// :Description: Example function block for TcKit parser validation.
// :param bEnable: Rising edge starts the operation
// :param nSetpoint: Target value in engineering units
FUNCTION_BLOCK FB_Example
VAR_INPUT
    bEnable    : BOOL;
    nSetpoint  : INT;
END_VAR
VAR_OUTPUT
    bDone      : BOOL;
    bError     : BOOL;
    nErrorId   : UDINT;
END_VAR
VAR
    eState     : E_ExampleState := E_ExampleState.Idle;
    nInternal  : INT;
END_VAR


CASE eState OF
    E_ExampleState.Idle:
        IF bEnable THEN
            eState := E_ExampleState.Running;
        END_IF

    E_ExampleState.Running:
        nInternal := nSetpoint;
        bDone := TRUE;
        eState := E_ExampleState.Idle;

    E_ExampleState.Error:
        bError := TRUE;
END_CASE


// :Description: Execute one cycle of the operation.
// :returns: TRUE when the operation completes successfully
METHOD Execute : BOOL
VAR_INPUT
    bTrigger : BOOL;
END_VAR

IF bTrigger THEN
    bDone := FALSE;
    bError := FALSE;
    nErrorId := 0;
    eState := E_ExampleState.Running;
END_IF

Execute := bDone;
END_METHOD


// :Description: Reset error state and outputs.
METHOD Reset : BOOL

bDone := FALSE;
bError := FALSE;
nErrorId := 0;
eState := E_ExampleState.Idle;
Reset := TRUE;
END_METHOD

END_FUNCTION_BLOCK

(* stored: Version 1.1.0.1, ProductVersion 3.1.4026.0
   POU FB_Example: Id {12345678-0000-0000-0000-000000000001}, SpecialFunc None
   Method Execute: Id {12345678-0000-0000-0000-000000000002}
   Method Reset: Id {12345678-0000-0000-0000-000000000003} *)
